% RSLogix 500 project PV72.RSS, saved by version 8.30.00.16 %
PROJECT "PV72"    % processor: Bul.1763 MicroLogix 1100 Series B %

PROGRAM FILES
  LAD 2   37 rungs

DATA FILES
  O0 OUTPUT  6 elements
  I1 INPUT  7 elements
  S2 STATUS  66 elements
  B3 BINARY  3 elements
  T4 TIMER  3 elements
  C5 COUNTER  1 elements
  R6 CONTROL  1 elements
  N7 INTEGER  1 elements
  F8 FLOAT  1 elements

LADDER 2
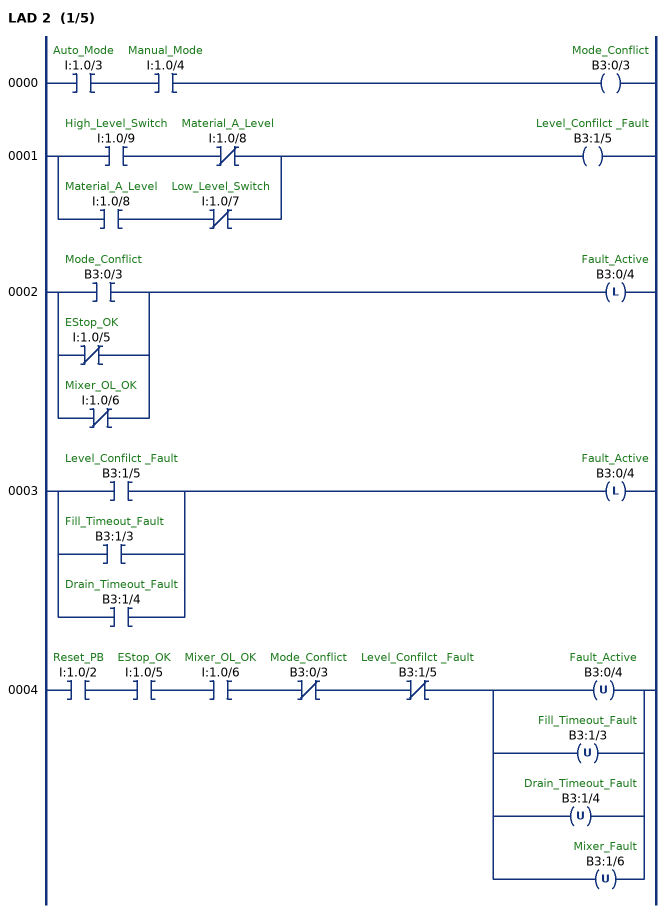
% Rung: 0 %
SOR XIC I:1.0/3 XIC I:1.0/4 OTE B3:0/3 EOR
%   I:1.0/3  "Auto_Mode" %
%   I:1.0/4  "Manual_Mode" %
%   B3:0/3  "Mode_Conflict" %
% Rung: 1 %
SOR BST XIC I:1.0/9 XIO I:1.0/8 NXB XIC I:1.0/8 XIO I:1.0/7 BND OTE B3:1/5 EOR
%   I:1.0/9  "High_Level_Switch" %
%   I:1.0/8  "Material_A_Level" %
%   I:1.0/7  "Low_Level_Switch" %
%   B3:1/5  "Level_Confilct _Fault" %
% Rung: 2 %
SOR BST XIC B3:0/3 NXB BST XIO I:1.0/5 NXB XIO I:1.0/6 BND BND OTL B3:0/4 EOR
%   B3:0/3  "Mode_Conflict" %
%   I:1.0/5  "EStop_OK" %
%   I:1.0/6  "Mixer_OL_OK" %
%   B3:0/4  "Fault_Active" %
% Rung: 3 %
SOR BST XIC B3:1/5 NXB BST XIC B3:1/3 NXB XIC B3:1/4 BND BND OTL B3:0/4 EOR
%   B3:1/5  "Level_Confilct _Fault" %
%   B3:1/3  "Fill_Timeout_Fault" %
%   B3:1/4  "Drain_Timeout_Fault" %
%   B3:0/4  "Fault_Active" %
% Rung: 4 %
SOR XIC I:1.0/2 XIC I:1.0/5 XIC I:1.0/6 XIO B3:0/3 XIO B3:1/5 BST OTU B3:0/4 NXB BST OTU B3:1/3 NXB BST OTU B3:1/4 NXB OTU B3:1/6 BND BND BND EOR
%   I:1.0/2  "Reset_PB" %
%   I:1.0/5  "EStop_OK" %
%   I:1.0/6  "Mixer_OL_OK" %
%   B3:0/3  "Mode_Conflict" %
%   B3:1/5  "Level_Confilct _Fault" %
%   B3:0/4  "Fault_Active" %
%   B3:1/3  "Fill_Timeout_Fault" %
%   B3:1/4  "Drain_Timeout_Fault" %
%   B3:1/6  "Mixer_Fault" %

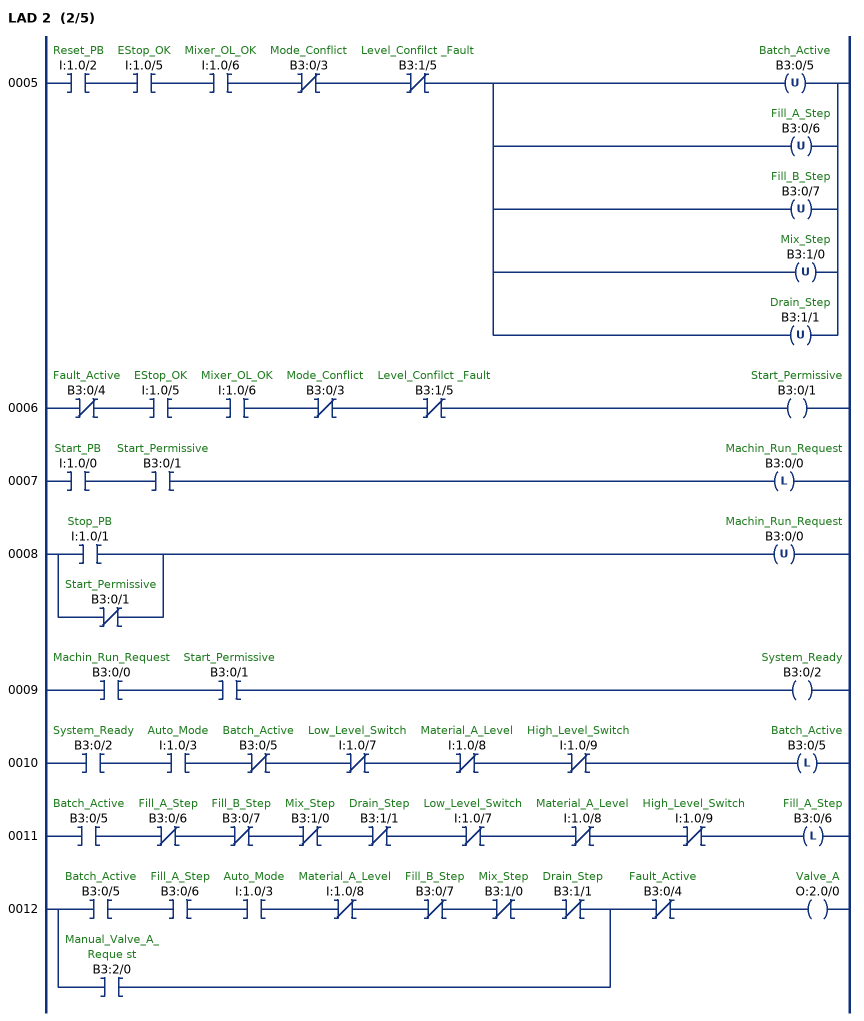
% Rung: 5 %
SOR XIC I:1.0/2 XIC I:1.0/5 XIC I:1.0/6 XIO B3:0/3 XIO B3:1/5 BST OTU B3:0/5 NXB BST OTU B3:0/6 NXB BST OTU B3:0/7 NXB BST OTU B3:1/0 NXB OTU B3:1/1 BND BND BND BND EOR
%   I:1.0/2  "Reset_PB" %
%   I:1.0/5  "EStop_OK" %
%   I:1.0/6  "Mixer_OL_OK" %
%   B3:0/3  "Mode_Conflict" %
%   B3:1/5  "Level_Confilct _Fault" %
%   B3:0/5  "Batch_Active" %
%   B3:0/6  "Fill_A_Step" %
%   B3:0/7  "Fill_B_Step" %
%   B3:1/0  "Mix_Step" %
%   B3:1/1  "Drain_Step" %
% Rung: 6 %
SOR XIO B3:0/4 XIC I:1.0/5 XIC I:1.0/6 XIO B3:0/3 XIO B3:1/5 OTE B3:0/1 EOR
%   B3:0/4  "Fault_Active" %
%   I:1.0/5  "EStop_OK" %
%   I:1.0/6  "Mixer_OL_OK" %
%   B3:0/3  "Mode_Conflict" %
%   B3:1/5  "Level_Confilct _Fault" %
%   B3:0/1  "Start_Permissive" %
% Rung: 7 %
SOR XIC I:1.0/0 XIC B3:0/1 OTL B3:0/0 EOR
%   I:1.0/0  "Start_PB" %
%   B3:0/1  "Start_Permissive" %
%   B3:0/0  "Machin_Run_Request" %
% Rung: 8 %
SOR BST XIC I:1.0/1 NXB XIO B3:0/1 BND OTU B3:0/0 EOR
%   I:1.0/1  "Stop_PB" %
%   B3:0/1  "Start_Permissive" %
%   B3:0/0  "Machin_Run_Request" %
% Rung: 9 %
SOR XIC B3:0/0 XIC B3:0/1 OTE B3:0/2 EOR
%   B3:0/0  "Machin_Run_Request" %
%   B3:0/1  "Start_Permissive" %
%   B3:0/2  "System_Ready" %
% Rung: 10 %
SOR XIC B3:0/2 XIC I:1.0/3 XIO B3:0/5 XIO I:1.0/7 XIO I:1.0/8 XIO I:1.0/9 OTL B3:0/5 EOR
%   B3:0/2  "System_Ready" %
%   I:1.0/3  "Auto_Mode" %
%   B3:0/5  "Batch_Active" %
%   I:1.0/7  "Low_Level_Switch" %
%   I:1.0/8  "Material_A_Level" %
%   I:1.0/9  "High_Level_Switch" %
% Rung: 11 %
SOR XIC B3:0/5 XIO B3:0/6 XIO B3:0/7 XIO B3:1/0 XIO B3:1/1 XIO I:1.0/7 XIO I:1.0/8 XIO I:1.0/9 OTL B3:0/6 EOR
%   B3:0/5  "Batch_Active" %
%   B3:0/6  "Fill_A_Step" %
%   B3:0/7  "Fill_B_Step" %
%   B3:1/0  "Mix_Step" %
%   B3:1/1  "Drain_Step" %
%   I:1.0/7  "Low_Level_Switch" %
%   I:1.0/8  "Material_A_Level" %
%   I:1.0/9  "High_Level_Switch" %
% Rung: 12 %
SOR BST XIC B3:0/5 XIC B3:0/6 XIC I:1.0/3 XIO I:1.0/8 XIO B3:0/7 XIO B3:1/0 XIO B3:1/1 NXB XIC B3:2/0 BND XIO B3:0/4 OTE O:2.0/0 EOR
%   B3:0/5  "Batch_Active" %
%   B3:0/6  "Fill_A_Step" %
%   I:1.0/3  "Auto_Mode" %
%   I:1.0/8  "Material_A_Level" %
%   B3:0/7  "Fill_B_Step" %
%   B3:1/0  "Mix_Step" %
%   B3:1/1  "Drain_Step" %
%   B3:2/0  "Manual_Valve_A_Reque st" %
%   B3:0/4  "Fault_Active" %
%   O:2.0/0  "Valve_A" %

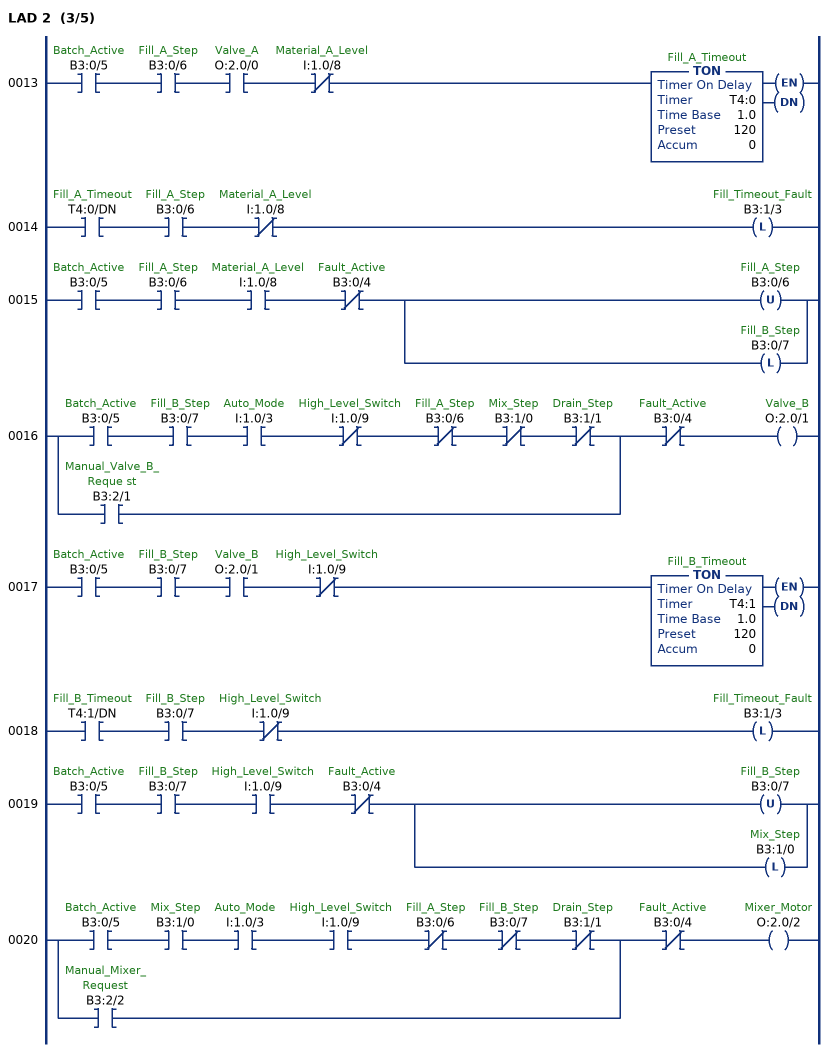
% Rung: 13 %
SOR XIC B3:0/5 XIC B3:0/6 XIC O:2.0/0 XIO I:1.0/8 TON T4:0 1.0 120 0 EOR
%   B3:0/5  "Batch_Active" %
%   B3:0/6  "Fill_A_Step" %
%   O:2.0/0  "Valve_A" %
%   I:1.0/8  "Material_A_Level" %
%   T4:0  "Fill_A_Timeout" %
% Rung: 14 %
SOR XIC T4:0/DN XIC B3:0/6 XIO I:1.0/8 OTL B3:1/3 EOR
%   T4:0  "Fill_A_Timeout" %
%   B3:0/6  "Fill_A_Step" %
%   I:1.0/8  "Material_A_Level" %
%   B3:1/3  "Fill_Timeout_Fault" %
% Rung: 15 %
SOR XIC B3:0/5 XIC B3:0/6 XIC I:1.0/8 XIO B3:0/4 BST OTU B3:0/6 NXB OTL B3:0/7 BND EOR
%   B3:0/5  "Batch_Active" %
%   B3:0/6  "Fill_A_Step" %
%   I:1.0/8  "Material_A_Level" %
%   B3:0/4  "Fault_Active" %
%   B3:0/7  "Fill_B_Step" %
% Rung: 16 %
SOR BST XIC B3:0/5 XIC B3:0/7 XIC I:1.0/3 XIO I:1.0/9 XIO B3:0/6 XIO B3:1/0 XIO B3:1/1 NXB XIC B3:2/1 BND XIO B3:0/4 OTE O:2.0/1 EOR
%   B3:0/5  "Batch_Active" %
%   B3:0/7  "Fill_B_Step" %
%   I:1.0/3  "Auto_Mode" %
%   I:1.0/9  "High_Level_Switch" %
%   B3:0/6  "Fill_A_Step" %
%   B3:1/0  "Mix_Step" %
%   B3:1/1  "Drain_Step" %
%   B3:2/1  "Manual_Valve_B_Reque st" %
%   B3:0/4  "Fault_Active" %
%   O:2.0/1  "Valve_B" %
% Rung: 17 %
SOR XIC B3:0/5 XIC B3:0/7 XIC O:2.0/1 XIO I:1.0/9 TON T4:1 1.0 120 0 EOR
%   B3:0/5  "Batch_Active" %
%   B3:0/7  "Fill_B_Step" %
%   O:2.0/1  "Valve_B" %
%   I:1.0/9  "High_Level_Switch" %
%   T4:1  "Fill_B_Timeout" %
% Rung: 18 %
SOR XIC T4:1/DN XIC B3:0/7 XIO I:1.0/9 OTL B3:1/3 EOR
%   T4:1  "Fill_B_Timeout" %
%   B3:0/7  "Fill_B_Step" %
%   I:1.0/9  "High_Level_Switch" %
%   B3:1/3  "Fill_Timeout_Fault" %
% Rung: 19 %
SOR XIC B3:0/5 XIC B3:0/7 XIC I:1.0/9 XIO B3:0/4 BST OTU B3:0/7 NXB OTL B3:1/0 BND EOR
%   B3:0/5  "Batch_Active" %
%   B3:0/7  "Fill_B_Step" %
%   I:1.0/9  "High_Level_Switch" %
%   B3:0/4  "Fault_Active" %
%   B3:1/0  "Mix_Step" %
% Rung: 20 %
SOR BST XIC B3:0/5 XIC B3:1/0 XIC I:1.0/3 XIC I:1.0/9 XIO B3:0/6 XIO B3:0/7 XIO B3:1/1 NXB XIC B3:2/2 BND XIO B3:0/4 OTE O:2.0/2 EOR
%   B3:0/5  "Batch_Active" %
%   B3:1/0  "Mix_Step" %
%   I:1.0/3  "Auto_Mode" %
%   I:1.0/9  "High_Level_Switch" %
%   B3:0/6  "Fill_A_Step" %
%   B3:0/7  "Fill_B_Step" %
%   B3:1/1  "Drain_Step" %
%   B3:2/2  "Manual_Mixer_Request" %
%   B3:0/4  "Fault_Active" %
%   O:2.0/2  "Mixer_Motor" %

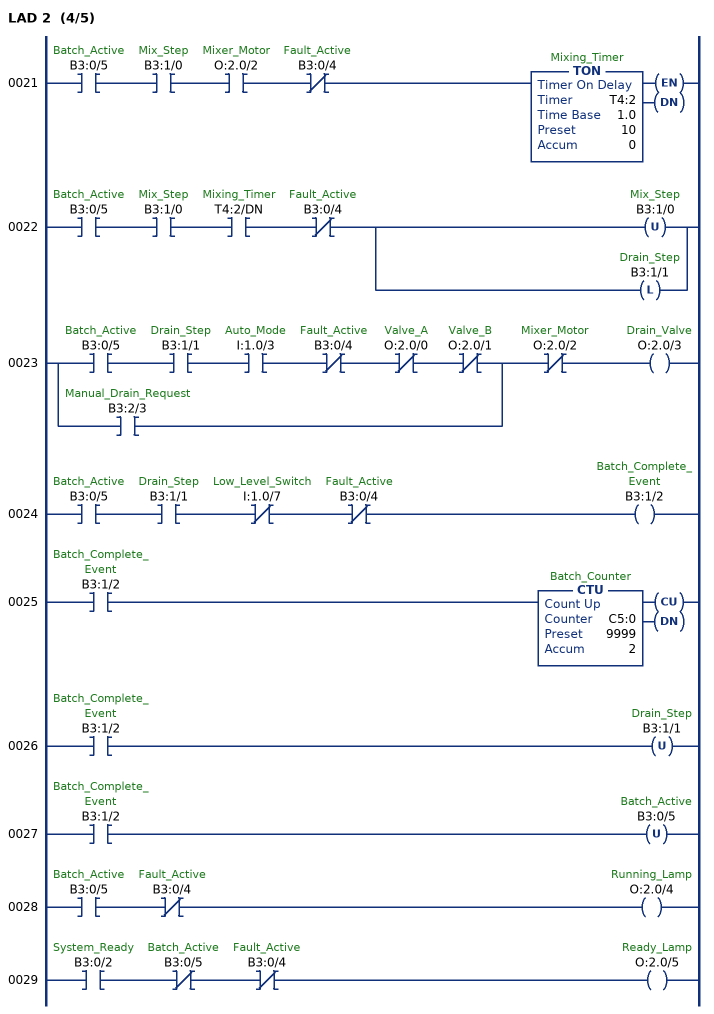
% Rung: 21 %
SOR XIC B3:0/5 XIC B3:1/0 XIC O:2.0/2 XIO B3:0/4 TON T4:2 1.0 10 0 EOR
%   B3:0/5  "Batch_Active" %
%   B3:1/0  "Mix_Step" %
%   O:2.0/2  "Mixer_Motor" %
%   B3:0/4  "Fault_Active" %
%   T4:2  "Mixing_Timer" %
% Rung: 22 %
SOR XIC B3:0/5 XIC B3:1/0 XIC T4:2/DN XIO B3:0/4 BST OTU B3:1/0 NXB OTL B3:1/1 BND EOR
%   B3:0/5  "Batch_Active" %
%   B3:1/0  "Mix_Step" %
%   T4:2  "Mixing_Timer" %
%   B3:0/4  "Fault_Active" %
%   B3:1/1  "Drain_Step" %
% Rung: 23 %
SOR BST XIC B3:0/5 XIC B3:1/1 XIC I:1.0/3 XIO B3:0/4 XIO O:2.0/0 XIO O:2.0/1 NXB XIC B3:2/3 BND XIO O:2.0/2 OTE O:2.0/3 EOR
%   B3:0/5  "Batch_Active" %
%   B3:1/1  "Drain_Step" %
%   I:1.0/3  "Auto_Mode" %
%   B3:0/4  "Fault_Active" %
%   O:2.0/0  "Valve_A" %
%   O:2.0/1  "Valve_B" %
%   B3:2/3  "Manual_Drain_Request" %
%   O:2.0/2  "Mixer_Motor" %
%   O:2.0/3  "Drain_Valve" %
% Rung: 24 %
SOR XIC B3:0/5 XIC B3:1/1 XIO I:1.0/7 XIO B3:0/4 OTE B3:1/2 EOR
%   B3:0/5  "Batch_Active" %
%   B3:1/1  "Drain_Step" %
%   I:1.0/7  "Low_Level_Switch" %
%   B3:0/4  "Fault_Active" %
%   B3:1/2  "Batch_Complete_Event" %
% Rung: 25 %
SOR XIC B3:1/2 CTU C5:0 9999 2 EOR
%   B3:1/2  "Batch_Complete_Event" %
%   C5:0  "Batch_Counter" %
% Rung: 26 %
SOR XIC B3:1/2 OTU B3:1/1 EOR
%   B3:1/2  "Batch_Complete_Event" %
%   B3:1/1  "Drain_Step" %
% Rung: 27 %
SOR XIC B3:1/2 OTU B3:0/5 EOR
%   B3:1/2  "Batch_Complete_Event" %
%   B3:0/5  "Batch_Active" %
% Rung: 28 %
SOR XIC B3:0/5 XIO B3:0/4 OTE O:2.0/4 EOR
%   B3:0/5  "Batch_Active" %
%   B3:0/4  "Fault_Active" %
%   O:2.0/4  "Running_Lamp" %
% Rung: 29 %
SOR XIC B3:0/2 XIO B3:0/5 XIO B3:0/4 OTE O:2.0/5 EOR
%   B3:0/2  "System_Ready" %
%   B3:0/5  "Batch_Active" %
%   B3:0/4  "Fault_Active" %
%   O:2.0/5  "Ready_Lamp" %

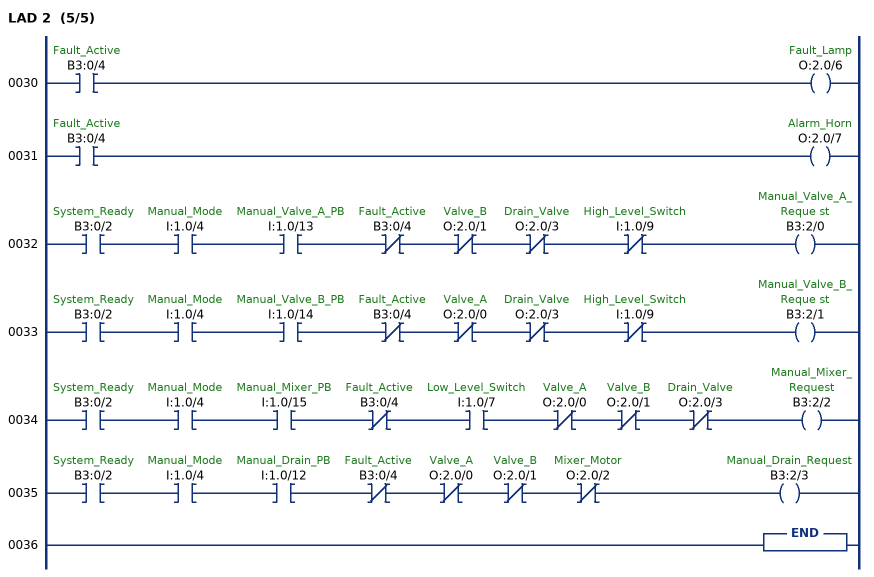
% Rung: 30 %
SOR XIC B3:0/4 OTE O:2.0/6 EOR
%   B3:0/4  "Fault_Active" %
%   O:2.0/6  "Fault_Lamp" %
% Rung: 31 %
SOR XIC B3:0/4 OTE O:2.0/7 EOR
%   B3:0/4  "Fault_Active" %
%   O:2.0/7  "Alarm_Horn" %
% Rung: 32 %
SOR XIC B3:0/2 XIC I:1.0/4 XIC I:1.0/13 XIO B3:0/4 XIO O:2.0/1 XIO O:2.0/3 XIO I:1.0/9 OTE B3:2/0 EOR
%   B3:0/2  "System_Ready" %
%   I:1.0/4  "Manual_Mode" %
%   I:1.0/13  "Manual_Valve_A_PB" %
%   B3:0/4  "Fault_Active" %
%   O:2.0/1  "Valve_B" %
%   O:2.0/3  "Drain_Valve" %
%   I:1.0/9  "High_Level_Switch" %
%   B3:2/0  "Manual_Valve_A_Reque st" %
% Rung: 33 %
SOR XIC B3:0/2 XIC I:1.0/4 XIC I:1.0/14 XIO B3:0/4 XIO O:2.0/0 XIO O:2.0/3 XIO I:1.0/9 OTE B3:2/1 EOR
%   B3:0/2  "System_Ready" %
%   I:1.0/4  "Manual_Mode" %
%   I:1.0/14  "Manual_Valve_B_PB" %
%   B3:0/4  "Fault_Active" %
%   O:2.0/0  "Valve_A" %
%   O:2.0/3  "Drain_Valve" %
%   I:1.0/9  "High_Level_Switch" %
%   B3:2/1  "Manual_Valve_B_Reque st" %
% Rung: 34 %
SOR XIC B3:0/2 XIC I:1.0/4 XIC I:1.0/15 XIO B3:0/4 XIC I:1.0/7 XIO O:2.0/0 XIO O:2.0/1 XIO O:2.0/3 OTE B3:2/2 EOR
%   B3:0/2  "System_Ready" %
%   I:1.0/4  "Manual_Mode" %
%   I:1.0/15  "Manual_Mixer_PB" %
%   B3:0/4  "Fault_Active" %
%   I:1.0/7  "Low_Level_Switch" %
%   O:2.0/0  "Valve_A" %
%   O:2.0/1  "Valve_B" %
%   O:2.0/3  "Drain_Valve" %
%   B3:2/2  "Manual_Mixer_Request" %
% Rung: 35 %
SOR XIC B3:0/2 XIC I:1.0/4 XIC I:1.0/12 XIO B3:0/4 XIO O:2.0/0 XIO O:2.0/1 XIO O:2.0/2 OTE B3:2/3 EOR
%   B3:0/2  "System_Ready" %
%   I:1.0/4  "Manual_Mode" %
%   I:1.0/12  "Manual_Drain_PB" %
%   B3:0/4  "Fault_Active" %
%   O:2.0/0  "Valve_A" %
%   O:2.0/1  "Valve_B" %
%   O:2.0/2  "Mixer_Motor" %
%   B3:2/3  "Manual_Drain_Request" %
% Rung: 36 %
SOR END EOR

DATA TABLE (non-zero values as saved)
DATA B3
% B3:0 % 0X0010 0X0000 0X0000
DATA T4
% .PRE .ACC %
% T4:0 % 120 0
% T4:1 % 120 0
% T4:2 % 10 0
DATA C5
% .PRE .ACC %
% C5:0 % 9999 2
